// TIA Portal V18 export
// export: Created 2025-12-01T12:39:34.9509233Z, ExportSetting None, DisplayName Totally Integrated Automation Portal, DisplayVersion V18 Update 5, DisplayName TIA Portal Openness, DisplayVersion V18 Update 5, DisplayName TIA Portal Teamcenter Gateway, DisplayVersion V18, DisplayName TIA Portal Version Control Interface, DisplayVersion V18, DisplayName STEP 7 Professional, DisplayVersion V18 Update 5, DisplayName STEP 7 Safety, DisplayVersion V18, DisplayName WinCC Professional, DisplayVersion V18 Update 5
VAR_GLOBAL   // PLC tag table "PLCIO_DI"
   "iHMI Control On" AT %I100.0 : Bool;   // HMI_上电按钮
   "iHMI Machine Start" AT %I100.1 : Bool;   // HMI_设备启动按钮
   "iHMI Machine Stop" AT %I100.2 : Bool;   // HMI_设备停止按钮
   "iHMI ResetButton" AT %I100.3 : Bool;   // HMI_复位按钮
   "iHMI Manual/Auto" AT %I100.4 : Bool;   // HMI_手/自动切换按钮
   "iHMI Safety Gate Unlock" AT %I100.5 : Bool;   // HMI_安全门解锁按钮
   "iHMI E-Stop" AT %I100.6 : Bool;   // HMI_急停
   "iRESERVE_I100.7" AT %I100.7 : Bool;   // 备用_I100.7
   iPressure AT %I101.0 : Bool;   // 气压监控
   "iCircuit Breaker OK_1" AT %I101.1 : Bool;   // 电子断路器 OK_1
   "iCircuit Breaker OK_2" AT %I101.2 : Bool;   // 电子断路器 OK_2
   "iRESERVE_I101.3" AT %I101.3 : Bool;   // 备用_I101.3
   iE_StopButton2_A01 AT %I101.4 : Bool;   // A01急停按钮2
   iNG_Button1 AT %I101.5 : Bool;   // NG下料按钮1
   iE_StopButton3_A02 AT %I101.6 : Bool;   // A02急停按钮3
   iNG_Button2 AT %I101.7 : Bool;   // NG下料按钮2
   "iSafety door Locking FeedBack_1" AT %I102.0 : Bool;   // 安全门锁定反馈_1
   "iSafety door Locking FeedBack_2" AT %I102.1 : Bool;   // 安全门锁定反馈_2
   "iSafety door Locking FeedBack_3" AT %I102.2 : Bool;   // 安全门锁定反馈_3
   "iSafety door Locking FeedBack_4" AT %I102.3 : Bool;   // 安全门锁定反馈_4
   "iSafety door Locking FeedBack_5" AT %I102.4 : Bool;   // 安全门锁定反馈_5
   "iSafety door Locking FeedBack_6" AT %I102.5 : Bool;   // 安全门锁定反馈_6
   "iSafety door Locking FeedBack_7" AT %I102.6 : Bool;   // 安全门锁定反馈_7
   "iSafety door Locking FeedBack_8" AT %I102.7 : Bool;   // 安全门锁定反馈_8
   "iSafety Door Locking FeedBack" AT %I103.0 : Bool;   // 连锁安全门锁定反馈
   "iMateriel Door Locking FeedBack_H1" AT %I103.1 : Bool;   // 物料门锁定反馈_1
   "iMateriel Door Locking FeedBack_H2" AT %I103.2 : Bool;   // 物料门锁定反馈_2
   "iMateriel Door Locking FeedBack_J1" AT %I103.3 : Bool;   // 物料门锁定反馈_3
   "iMateriel Door Locking FeedBack_J2" AT %I103.4 : Bool;   // 物料门锁定反馈_4
   "iMateriel Door Locking FeedBack_K1" AT %I103.5 : Bool;   // 物料门锁定反馈_5
   "iMateriel Door Locking FeedBack_K2" AT %I103.6 : Bool;   // 物料门锁定反馈_6
   "iMateriel Door Locking FeedBack_L1" AT %I103.7 : Bool;   // 物料门锁定反馈_7
   iShaft_Button AT %I104.1 : Bool;   // shaft 上料按钮
   iE_StopButton4_H AT %I104.0 : Bool;   // H_急停按钮4
   iShaft_EmptyButton AT %I104.2 : Bool;   // shaft 取空料盘按钮
   iE_StopButton5_J AT %I104.3 : Bool;   // J_急停按钮5
   iMagnet_Button AT %I104.4 : Bool;   // Magnet上料按钮
   iMagnet_EmptyButton AT %I104.5 : Bool;   // Magnet取空料盘按钮
   iMagnet_UnlockButton AT %I104.6 : Bool;   // Magne门解锁按钮
   "iRESERVE_I104.7" AT %I104.7 : Bool;   // 备用_I104.7
   iE_StopButton6_K AT %I105.0 : Bool;   // K_急停按钮6
   iReserved_Button AT %I105.1 : Bool;   // Reserved上料按钮
   iReserved_EmptyButton AT %I105.2 : Bool;   // Reserved取空料盘按钮
   iReserved_UnlockButton AT %I105.3 : Bool;   // Reserved门解锁按钮
   iE_StopButton7_L AT %I105.4 : Bool;   // L_急停按钮7
   iUnloading_Button AT %I105.5 : Bool;   // Unloading按钮
   iUnloading_EmptyButton AT %I105.6 : Bool;   // Unloading取空料盘按钮
   iUnloading_UnlockButton AT %I105.7 : Bool;   // Unloading门解锁按钮
   "iE-NG-01 Safety Gate_Open" AT %I106.0 : Bool;   // E-NG料盒-01安全门锁_a
   "iE-NG-01 Safety Gate_UnLock" AT %I106.1 : Bool;   // E-NG料盒-01安全门锁_b
   "iE-NG-02 Safety Gate_Open" AT %I106.2 : Bool;   // E-NG料盒-02安全门锁_a
   "iE-NG-02 Safety Gate_UnLock" AT %I106.3 : Bool;   // E-NG料盒-02安全门锁_b
   iALightCurtain_1 AT %I106.4 : Bool;   // 备用_I106.4 / A-光栅1
   iALightCurtain_2 AT %I106.5 : Bool;   // 备用_I106.5 / A-光栅2
   "iRESERVE_I106.6" AT %I106.6 : Bool;   // 备用_I106.6
   "iRESERVE_I106.7" AT %I106.7 : Bool;   // 备用_I106.7
   "iH-shaft Loading _a" AT %I107.0 : Bool;   // H-shaft上料线体驱动电机_a
   "iH-shaft Loading _b" AT %I107.1 : Bool;   // H-shaft上料线体驱动电机_b
   "iH-shaft Take _a" AT %I107.2 : Bool;   // H-shaft取空盘驱动电机_a
   "iH-shaft Take _b" AT %I107.3 : Bool;   // H-shaft取空盘驱动电机_b
   "iH-shaft  Lifting _a" AT %I107.4 : Bool;   // H-shaft 顶升位驱动电机_a
   "iH-shaft  Lifting _b" AT %I107.5 : Bool;   // H-shaft 顶升位驱动电机_b
   "iRESERVE_I107.6" AT %I107.6 : Bool;   // 备用_I107.6
   "iRESERVE_I107.7" AT %I107.7 : Bool;   // 备用_I107.7
   "iJ-magnet Loading _a" AT %I108.0 : Bool;   // J-magnet上料线体驱动电机_a
   "iJ-magnet Loading _b" AT %I108.1 : Bool;   // J-magnet上料线体驱动电机_b
   "iJ-magnet Take _a" AT %I108.2 : Bool;   // J-magnet取空盘驱动电机_a
   "iJ-magnet Take _b" AT %I108.3 : Bool;   // J-magnet取空盘驱动电机_b
   "iJ-magnet Lifting _a" AT %I108.4 : Bool;   // J-magnet顶升驱动电机_a
   "iJ-magnet Lifting _b" AT %I108.5 : Bool;   // J-magnet顶升驱动电机_b
   "iRESERVE_I108.6" AT %I108.6 : Bool;   // 备用_I108.6
   "iRESERVE_I108.7" AT %I108.7 : Bool;   // 备用_I108.7
   "iK-reserve Loading _a" AT %I109.0 : Bool;   // K-预留上料线体驱动电机_a
   "iK-reserve Loading _b" AT %I109.1 : Bool;   // K-预留上料线体驱动电机_b
   "iK-reserve Take _a" AT %I109.2 : Bool;   // K-预留取空盘驱动电机_a
   "iK-reserve Take _b" AT %I109.3 : Bool;   // K-预留取空盘驱动电机_b
   "iK-reserve Lifting3 _a" AT %I109.4 : Bool;   // K-预留顶升位3驱动电机_a
   "iK-reserve Lifting3 _b" AT %I109.5 : Bool;   // K-预留顶升位3驱动电机_b
   "iRESERVE_I109.6" AT %I109.6 : Bool;   // 备用_I109.6
   "iRESERVE_I109.7" AT %I109.7 : Bool;   // 备用_I109.7
   "iC- GluingDeviceReady" AT %I110.0 : Bool;   // C-涂胶模组点胶阀_a / C-涂胶系统准备就绪
   "iC- GluingFault" AT %I110.1 : Bool;   // C-涂胶模组点胶阀_b / C-涂胶系统报错
   "iC- GluingRefillTank" AT %I110.2 : Bool;   // C-涂胶模组点胶阀_c / C-涂胶系统缺料
   "iC- GluingTankEmpty" AT %I110.3 : Bool;   // 备用_I110.3 / C-涂胶系统空料
   "iL-Unloading Drive motor_a" AT %I110.4 : Bool;   // L-下料线体驱动电机_a
   "iL-Unloading Drive motor_b" AT %I110.5 : Bool;   // L-下料线体驱动电机_b
   "iL-Unloading transplanting motor_a" AT %I110.6 : Bool;   // L-下料线体移栽电机_a
   "iL-Unloading transplanting motor_b" AT %I110.7 : Bool;   // L-下料线体移栽电机_b
   iH_StopButton AT %I111.0 : Bool;
   iJ_StopButton AT %I111.1 : Bool;
   iK_StopButton AT %I111.2 : Bool;
   "iRESERVE_I111.3" AT %I111.3 : Bool;
   "iRESERVE_I111.4" AT %I111.4 : Bool;
   "iRESERVE_I111.5" AT %I111.5 : Bool;
   "iRESERVE_I111.6" AT %I111.6 : Bool;
   "iRESERVE_I111.7" AT %I111.7 : Bool;
END_VAR
